(* IEC 61131-3 sources: TCP_Data_Decode_For_plc/, 5 files *)

(* ---- CSV TCPIP Control.ST ---- *)
(* Get Date Time Stamp Now *)
s_Local_DateTimeNow	:= Replace(s_DateTimeNow,'',3,1);				// Trim awat DT# from Date time Stamp String

gb_Trig_TCPIP_Wr_Data_Write:= bSendingToClient_SvrID_1;

(*Compute Message*)
b_OneShot[45](CLK:= gb_Trig_TCPIP_Rec_Data_Write );
IF b_OneShot[45].Q THEN

	m1i	:= 1;			// Set Start Message Pointer to 1

			(* Part  Data Message  *)
			_s_TCPIP_Rec_CSVData_Message[m1i]:=Concat(s_Local_DateTimeNow	 ,',');
			_s_TCPIP_Rec_CSVData_Message[m1i]:=Concat(_s_TCPIP_Rec_CSVData_Message[mi],sFromClient_Recd_at_Server_SvrID_2);

			gb_WriteCSV_TCPIPLogRecData:=TRUE;					// CSV Write TCPIP Send Data
			gb_Trig_TCPIP_Rec_Data_Write:=FALSE;				// Clear Request Compute and TCPIP Send Data Bit

END_IF

(*Compute Message*)
b_OneShot[46](CLK:= gb_Trig_TCPIP_Wr_Data_Write );
IF b_OneShot[46].Q THEN

	m1i	:= 1;			// Set Start Message Pointer to 1

			(* Part  Data Message  *)
			_s_TCPIP_Wr_CSVData_Message[m1i]:=Concat(s_Local_DateTimeNow	 ,',');
			_s_TCPIP_Wr_CSVData_Message[m1i]:=Concat(_s_TCPIP_Wr_CSVData_Message[mi],strToClient_from_Server_SvrID_1);

			gb_WriteCSV_TCPIPLogWrData:=TRUE;					// CSV Write TCPIP Send Data
			gb_Trig_TCPIP_Wr_Data_Write:=FALSE;				// Clear Request Compute and TCPIP Send Data Bit

END_IF

(* ---- Declaration.ST ---- *)
PROGRAM Base_TcpIP_DecodenData
VAR

(* Decode Result Work Variable*)
s_IdentString			: ARRAY[1..30] OF T_MaxString;
 s_EndStringIdent1		: STRING[2] :='&';
 s_EndStringIdent2		: STRING[2] :='$$';

 s_DecodeString			: ARRAY[1..30] OF  T_MaxString;

 s_TrimStringData		:  T_MaxString;
 s_ReceivedString		:  T_MaxString;

 d_StartTrim_Index		: INT;
 d_NextTrim_Index		: INT;
 d_EndTrim_Index		: INT;

 d_HolderRef			: DINT;				// Current Holder Reference Number

 DataConfirm_Clk		:R_Trig;

 (* For Looping Variable*)

 ii			: INT :=1;
 xx			: INT :=1;

(* End Decode Result Variable*)

(* CSV Message & OPC Data Working Declaration*)

	mi									:INT :=1;				// Message Array Index Pointer
	m1i									:INT :=1;				// Message Array Index Pointer
	m2i									:INT :=1;				// Message Array Index Pointer
	m3i									:INT :=1;				// Message Array Index Pointer
	m4i									:INT :=1;				// Message Array Index Pointer

	s_Local_DateTimeNow					: String[22];
	b_OneShot 							:ARRAY [0..63]OF R_TRIG;	// 1 set of one shot Pulse bit for this module
	CD									:BOOL;						// Condition

(* End CSV Message & OPC Data Working Declaration*)
END_VAR

(* ---- Event Trigger Decoding.ST ---- *)
 DataConfirm_Clk(CLK:=isNewDataConfRecd_SvrID_2);

IF   DataConfirm_Clk.Q AND (LEN(sFromClient_Recd_at_Server_SvrID_2)>5) THEN

		gb_Trig_TCPIP_Rec_Data_Write		:=TRUE;				// Request TCPIP Log Received Data CSV
		R01_DecodeResult();										// Request Decode Received Data CSV
END_IF

(* ---- Output to CSV.ST ---- *)
(* Get Date Time Stamp Now *)
s_Local_DateTimeNow	:= Replace(s_DateTimeNow,'',3,1);				// Trim awat DT# from Date time Stamp String

(*Compute Message*)
b_OneShot[52](CLK:= gb_Trig_WeldData_Write );
IF b_OneShot[52].Q THEN

	mi	:= 1;			// Set Start Message Pointer to 1
	_s_WeldUnload_DMMC_Code:=_WeldDataArray[gd_HolderRef].dmcc;		// Copy The DMCC unload at Weld to Robot Arm

			(* Part  Data Message  *)
			_s_PartData_Weld_CSVData_Message[mi]:=Concat(s_Local_DateTimeNow	 ,',');
			_s_PartData_Weld_CSVData_Message[mi]:=Concat(_s_PartData_Weld_CSVData_Message[mi],DINT_TO_STRING(gd_HolderRef));
			_s_PartData_Weld_CSVData_Message[mi]:=Concat(_s_PartData_Weld_CSVData_Message[mi],',');
			_s_PartData_Weld_CSVData_Message[mi]:=Concat(_s_PartData_Weld_CSVData_Message[mi],DINT_TO_STRING(_WeldDataArray[gd_HolderRef].ttpos));
			_s_PartData_Weld_CSVData_Message[mi]:=Concat(_s_PartData_Weld_CSVData_Message[mi],',');
			_s_PartData_Weld_CSVData_Message[mi]:=Concat(_s_PartData_Weld_CSVData_Message[mi],(_WeldDataArray[gd_HolderRef].dmcc));
			_s_PartData_Weld_CSVData_Message[mi]:=Concat(_s_PartData_Weld_CSVData_Message[mi],',');
			_s_PartData_Weld_CSVData_Message[mi]:=Concat(_s_PartData_Weld_CSVData_Message[mi],DINT_TO_STRING(_WeldDataArray[gd_HolderRef].DataValue[4]));
			_s_PartData_Weld_CSVData_Message[mi]:=Concat(_s_PartData_Weld_CSVData_Message[mi],',');
			_s_PartData_Weld_CSVData_Message[mi]:=Concat(_s_PartData_Weld_CSVData_Message[mi],DINT_TO_STRING(_WeldDataArray[gd_HolderRef].DataValue[5]));
			_s_PartData_Weld_CSVData_Message[mi]:=Concat(_s_PartData_Weld_CSVData_Message[mi],',');
			_s_PartData_Weld_CSVData_Message[mi]:=Concat(_s_PartData_Weld_CSVData_Message[mi],DINT_TO_STRING(_WeldDataArray[gd_HolderRef].DataValue[6]));
			_s_PartData_Weld_CSVData_Message[mi]:=Concat(_s_PartData_Weld_CSVData_Message[mi],',');
			_s_PartData_Weld_CSVData_Message[mi]:=Concat(_s_PartData_Weld_CSVData_Message[mi],DINT_TO_STRING(_WeldDataArray[gd_HolderRef].DataValue[7]));
			_s_PartData_Weld_CSVData_Message[mi]:=Concat(_s_PartData_Weld_CSVData_Message[mi],',');
			_s_PartData_Weld_CSVData_Message[mi]:=Concat(_s_PartData_Weld_CSVData_Message[mi],DINT_TO_STRING(_WeldDataArray[gd_HolderRef].DataValue[8]));
			_s_PartData_Weld_CSVData_Message[mi]:=Concat(_s_PartData_Weld_CSVData_Message[mi],',');
			_s_PartData_Weld_CSVData_Message[mi]:=Concat(_s_PartData_Weld_CSVData_Message[mi],DINT_TO_STRING(_WeldDataArray[gd_HolderRef].DataValue[9]));
			_s_PartData_Weld_CSVData_Message[mi]:=Concat(_s_PartData_Weld_CSVData_Message[mi],',');
			_s_PartData_Weld_CSVData_Message[mi]:=Concat(_s_PartData_Weld_CSVData_Message[mi],DINT_TO_STRING(_WeldDataArray[gd_HolderRef].DataValue[10]));
			_s_PartData_Weld_CSVData_Message[mi]:=Concat(_s_PartData_Weld_CSVData_Message[mi],',');
			_s_PartData_Weld_CSVData_Message[mi]:=Concat(_s_PartData_Weld_CSVData_Message[mi],DINT_TO_STRING(_WeldDataArray[gd_HolderRef].DataValue[11]));
			_s_PartData_Weld_CSVData_Message[mi]:=Concat(_s_PartData_Weld_CSVData_Message[mi],',');
			_s_PartData_Weld_CSVData_Message[mi]:=Concat(_s_PartData_Weld_CSVData_Message[mi],DINT_TO_STRING(_WeldDataArray[gd_HolderRef].DataValue[12]));
			_s_PartData_Weld_CSVData_Message[mi]:=Concat(_s_PartData_Weld_CSVData_Message[mi],',');
			_s_PartData_Weld_CSVData_Message[mi]:=Concat(_s_PartData_Weld_CSVData_Message[mi],DINT_TO_STRING(_WeldDataArray[gd_HolderRef].DataValue[13]));
			_s_PartData_Weld_CSVData_Message[mi]:=Concat(_s_PartData_Weld_CSVData_Message[mi],',');
			_s_PartData_Weld_CSVData_Message[mi]:=Concat(_s_PartData_Weld_CSVData_Message[mi],DINT_TO_STRING(_WeldDataArray[gd_HolderRef].DataValue[14]));
			_s_PartData_Weld_CSVData_Message[mi]:=Concat(_s_PartData_Weld_CSVData_Message[mi],',');
			_s_PartData_Weld_CSVData_Message[mi]:=Concat(_s_PartData_Weld_CSVData_Message[mi],DINT_TO_STRING(_WeldDataArray[gd_HolderRef].DataValue[15]));
			_s_PartData_Weld_CSVData_Message[mi]:=Concat(_s_PartData_Weld_CSVData_Message[mi],',');
			_s_PartData_Weld_CSVData_Message[mi]:=Concat(_s_PartData_Weld_CSVData_Message[mi],DINT_TO_STRING(_WeldDataArray[gd_HolderRef].DataValue[16]));
			_s_PartData_Weld_CSVData_Message[mi]:=Concat(_s_PartData_Weld_CSVData_Message[mi],',');
			_s_PartData_Weld_CSVData_Message[mi]:=Concat(_s_PartData_Weld_CSVData_Message[mi],DINT_TO_STRING(_WeldDataArray[gd_HolderRef].DataValue[17]));
			_s_PartData_Weld_CSVData_Message[mi]:=Concat(_s_PartData_Weld_CSVData_Message[mi],',');
			_s_PartData_Weld_CSVData_Message[mi]:=Concat(_s_PartData_Weld_CSVData_Message[mi],DINT_TO_STRING(_WeldDataArray[gd_HolderRef].DataValue[18]));
			_s_PartData_Weld_CSVData_Message[mi]:=Concat(_s_PartData_Weld_CSVData_Message[mi],',');
			_s_PartData_Weld_CSVData_Message[mi]:=Concat(_s_PartData_Weld_CSVData_Message[mi],DINT_TO_STRING(_WeldDataArray[gd_HolderRef].DataValue[19]));
			_s_PartData_Weld_CSVData_Message[mi]:=Concat(_s_PartData_Weld_CSVData_Message[mi],',');
			_s_PartData_Weld_CSVData_Message[mi]:=Concat(_s_PartData_Weld_CSVData_Message[mi],DINT_TO_STRING(_WeldDataArray[gd_HolderRef].DataValue[20]));
			_s_PartData_Weld_CSVData_Message[mi]:=Concat(_s_PartData_Weld_CSVData_Message[mi],',');
			_s_PartData_Weld_CSVData_Message[mi]:=Concat(_s_PartData_Weld_CSVData_Message[mi],DINT_TO_STRING(_WeldDataArray[gd_HolderRef].DataValue[21]));
			_s_PartData_Weld_CSVData_Message[mi]:=Concat(_s_PartData_Weld_CSVData_Message[mi],',');
			_s_PartData_Weld_CSVData_Message[mi]:=Concat(_s_PartData_Weld_CSVData_Message[mi],DINT_TO_STRING(_WeldDataArray[gd_HolderRef].DataValue[22]));
			_s_PartData_Weld_CSVData_Message[mi]:=Concat(_s_PartData_Weld_CSVData_Message[mi],',');
			_s_PartData_Weld_CSVData_Message[mi]:=Concat(_s_PartData_Weld_CSVData_Message[mi],DINT_TO_STRING(_WeldDataArray[gd_HolderRef].DataValue[23]));
			_s_PartData_Weld_CSVData_Message[mi]:=Concat(_s_PartData_Weld_CSVData_Message[mi],',');
			_s_PartData_Weld_CSVData_Message[mi]:=Concat(_s_PartData_Weld_CSVData_Message[mi],DINT_TO_STRING(_WeldDataArray[gd_HolderRef].DataValue[24]));

			gd_UL_Hold_Result	:= _WeldDataArray[gd_HolderRef].DataValue[24];		// Copy Result Code to Galobal Tag
			gd_Prev_HoldRef		:= gd_HolderRef; 		// Set The Hold to Previous (For Record And Next Logging)
			gb_WriteCSV_WeldData:=TRUE;					// CSV Write weld Data
			gb_Trig_WeldData_Write:=FALSE;				// Clear Request Compute and Write Weld Data Bit

END_IF

(* ---- TCP decode.ST ---- *)
(* Decode String from TCP/IP Client*)

	// Defined Identification Keyword
	s_IdentString[1]			:= 'hold=';
	s_IdentString[2]			:= 'ttpos=';
	s_IdentString[3]			:= 'dmcc=';
	s_IdentString[4]			:= 'mvs1rl=';
	s_IdentString[5]			:= 'mvs1rr=';
	s_IdentString[6]			:= 'mvs1tl=';
	s_IdentString[7]			:= 'mvs1tr=';
	s_IdentString[8]			:= 'mvs3l=';
	s_IdentString[9]			:='mvs3r=';
	s_IdentString[10]			:='mvs71sl=';
	s_IdentString[11]			:='mvs71sr=';
	s_IdentString[12]			:='mvs71fl=';
	s_IdentString[13]			:='mvs71fr=';
	s_IdentString[14]			:='mvs3eclul=';
	s_IdentString[15]			:='mvs3ecldl=';
	s_IdentString[16]			:='mvs3eclur=';
	s_IdentString[17]			:='mvs3ecldr=';
	s_IdentString[18]			:='mvs3cul=';
	s_IdentString[19]			:='mvs3cur=';
	s_IdentString[20]			:='mvs3gul=';
	s_IdentString[21]			:='mvs3gur=';
	s_IdentString[22]			:='mvs6ptl=';
	s_IdentString[23]			:='mvs6ptr=';
	s_IdentString[24]			:='out=';
	s_IdentString[25]			:='error=';

															// sFromClient_Recd_at_Server_SvrID_2; 	// get String Data

	(*Find Identication Start String Index Number*)

FOR ii:=1 TO 30 BY 1 DO

	IF ii=1 THEN
			s_ReceivedString			:=sFromClient_Recd_at_Server_SvrID_2; 	// get String Data
			s_TrimStringData			:=s_ReceivedString;
	END_IF

	d_NextTrim_Index:=0;
	d_EndTrim_Index:=0;

	d_StartTrim_Index		:= FIND(s_TrimStringData,s_IdentString[ii]);
	IF d_StartTrim_Index>0 THEN

		s_TrimStringData		:= Delete (s_TrimStringData,(LEN(s_IdentString[ii])+(d_StartTrim_Index-1)),1);
		d_NextTrim_Index		:= FIND(s_TrimStringData,s_EndStringIdent1);
		 d_EndTrim_Index		:= FIND(s_TrimStringData,s_EndStringIdent2);

		 d_HolderRef			:= STRING_TO_DINT (s_DecodeString[1]);
		 gd_HolderRef			:=d_HolderRef;

		 IF d_NextTrim_Index>0 THEN
			 	s_DecodeString[ii]			:= MID(s_TrimStringData,d_NextTrim_Index-1,1);

				(* Get TTPOS to Weld Array Of the Holder*)
				IF ii=2 THEN
				_WeldDataArray[d_HolderRef].ttpos	:=STRING_TO_DINT(s_DecodeString[ii]);
				END_IF

				(* Get DMC String to Weld Array Of the Holder*)
				IF ii=3 THEN
				_WeldDataArray[d_HolderRef].DMCC	:=(s_DecodeString[ii]);
				END_IF

				(* Get Other String Data to Weld Array Of the Holder*)
				IF ii>=4 AND ii<=24 THEN
				_WeldDataArray[d_HolderRef].DataValue[ii]	:=STRING_TO_DINT(s_DecodeString[ii]);
				END_IF

				IF ii=25 THEN
				_WeldDataArray[d_HolderRef].error	:=s_DecodeString[ii];
				END_IF

		 END_IF

		 IF d_NextTrim_Index=0 THEN
			 	s_DecodeString[ii]		:= MID(s_TrimStringData,d_EndTrim_Index-1,1);

				IF ii>=4 AND ii<=24 THEN
				_WeldDataArray[d_HolderRef].DataValue[ii]	:=STRING_TO_DINT(s_DecodeString[ii]);
				END_IF

				IF ii=25 THEN
				_WeldDataArray[d_HolderRef].error	:=s_DecodeString[ii];
				END_IF

		 END_IF

	ELSE
 		IF (d_NextTrim_Index=0 AND d_EndTrim_Index=0) OR d_StartTrim_Index=0  THEN
			  	s_DecodeString[ii]		:= '';
		 END_IF

	  END_IF

	 gb_Trig_WeldData_Write:= (_WeldDataArray[d_HolderRef].ttpos =9);

END_FOR
